TYPE DUT_Struttura_Dati_Pacco :
STRUCT

	ID			: DUT_Lista_Pacchi_In_Pila;
	PC			: UINT;					(* Production Code *)
	PP      	: BOOL; 				(* Pack Presence *)

	X 			: REAL;					(* X dimension *)
	Y 			: REAL;					(* Y dimension *)
	Z 			: REAL;					(* Z dimension *)
	
END_STRUCT
END_TYPE

(* stored: Version 1.1.0.1, ProductVersion 3.1.4024.11
   DUT DUT_Struttura_Dati_Pacco: Id {3f71fd0c-4ee4-49a3-ac69-c6e5ba8f097c} *)
